{attribute 'GeneratedUsingTerminal: EP1518-0002-0016'}
{attribute addProperty BoxType "EP1518-0002-0016"}
{attribute addProperty Id "Set_counterBOOL1Inhibit_counterBOOL1"}
{attribute addProperty CRC "187665264"}
{attribute addProperty Size "2"}
TYPE Control_0B2F8B70 :
STRUCT
	{attribute addProperty Name "Set_counter"}
	Set_counter : BOOL;
	{attribute addProperty Name "Inhibit_counter"}
	Inhibit_counter : BOOL;
END_STRUCT
END_TYPE

(* stored: Version 1.2.0.0, ProductVersion 3.1.4024.9
   DUT Control_0B2F8B70: Id {c54745ae-5af0-40cc-836e-75747837e3c0} *)
